VISUALIZATION PneumaticCylinder  // 1024x768
END_VISUALIZATION

(* stored: Version 1.1.0.1, ProductVersion 3.1.4026.18
   Visu PneumaticCylinder: Id {48f56818-6056-4669-8f5b-90820557828c} *)
